# EPICS autosave request: SR570/iocBoot/iocstanfordSR570/auto_positions.req
file "XFM_SR570_positions.req",      P=XF:04BM-BMC:SR570, M={CurrAmp:1}
